FUNCTION_BLOCK aewaec
VAR_INPUT
END_VAR
VAR_OUTPUT
END_VAR
VAR
END_VAR

END_FUNCTION_BLOCK

(* stored: Version 1.1.0.1, ProductVersion 3.1.4020.12
   POU aewaec: Id {56e7f148-eb2d-43cc-bcdf-15eea7cd4097}, SpecialFunc None *)
